    movel([0.093526, -1.335742, -2.600974, -0.775673, 1.570796, 1.664322],accel_mss,speed_ms,0,blend_radius_m)
    movel([0.093093, -1.336352, -2.600581, -0.775456, 1.570796, 1.663890],accel_mss,speed_ms,0,blend_radius_m)
    movel([0.092892, -1.336973, -2.600181, -0.775235, 1.570796, 1.663688],accel_mss,speed_ms,0,blend_radius_m)
    movel([0.091818, -1.346006, -2.594298, -0.772085, 1.570796, 1.662615],accel_mss,speed_ms,0,blend_radius_m)
    movel([0.090858, -1.354768, -2.588485, -0.769136, 1.570796, 1.661654],accel_mss,speed_ms,0,blend_radius_m)
    movel([0.090901, -1.355470, -2.588015, -0.768904, 1.570796, 1.661698],accel_mss,speed_ms,0,blend_radius_m)
    movel([0.091183, -1.356047, -2.587628, -0.768714, 1.570796, 1.661979],accel_mss,speed_ms,0,blend_radius_m)
    movel([0.091406, -1.356179, -2.587539, -0.768671, 1.570796, 1.662202],accel_mss,speed_ms,0,blend_radius_m)
    movel([0.091721, -1.356174, -2.587542, -0.768673, 1.570796, 1.662517],accel_mss,speed_ms,0,blend_radius_m)
    movel([0.094111, -1.355583, -2.587939, -0.768867, 1.570796, 1.664908],accel_mss,speed_ms,0,blend_radius_m)
    movel([0.104155, -1.352656, -2.589896, -0.769837, 1.570796, 1.674951],accel_mss,speed_ms,0,blend_radius_m)
    movel([0.116814, -1.348919, -2.592378, -0.771092, 1.570796, 1.687610],accel_mss,speed_ms,0,blend_radius_m)
    movel([0.119225, -1.332381, -2.603128, -0.776879, 1.570796, 1.690022],accel_mss,speed_ms,0,blend_radius_m)
    movel([0.119516, -1.329656, -2.604864, -0.777869, 1.570796, 1.690312],accel_mss,speed_ms,0,blend_radius_m)
    movel([0.119518, -1.328189, -2.605795, -0.778406, 1.570796, 1.690314],accel_mss,speed_ms,0,blend_radius_m)
    movel([0.119398, -1.327925, -2.605961, -0.778502, 1.570796, 1.690195],accel_mss,speed_ms,0,blend_radius_m)
    movel([0.119109, -1.327817, -2.606030, -0.778542, 1.570796, 1.689905],accel_mss,speed_ms,0,blend_radius_m)
    movel([0.118012, -1.327865, -2.606000, -0.778525, 1.570796, 1.688809],accel_mss,speed_ms,0,blend_radius_m)
    movel([0.116851, -1.328114, -2.605842, -0.778433, 1.570796, 1.687647],accel_mss,speed_ms,0,blend_radius_m)
    movel([0.116553, -1.328203, -2.605786, -0.778400, 1.570796, 1.687349],accel_mss,speed_ms,0,blend_radius_m)
    speed_ms = 0.005
    movel([0.116553, -1.319188, -2.601551, -0.791650, 1.570796, 1.687349],accel_mss,speed_ms,0,blend_radius_m)
    speed_ms = 0.040
    movel([0.074162, -1.348204, -2.582858, -0.781327, 1.570796, 1.644958],accel_mss,speed_ms,0,blend_radius_m)
    speed_ms = 0.005
    movel([0.074162, -1.357034, -2.586964, -0.768391, 1.570796, 1.644958],accel_mss,speed_ms,0,blend_radius_m)
    speed_ms = 0.035
    movel([0.079007, -1.355499, -2.587996, -0.768895, 1.570796, 1.649804],accel_mss,speed_ms,0,blend_radius_m)
    movel([0.085319, -1.353347, -2.589435, -0.769607, 1.570796, 1.656115],accel_mss,speed_ms,0,blend_radius_m)
    movel([0.085564, -1.353072, -2.589619, -0.769698, 1.570796, 1.656361],accel_mss,speed_ms,0,blend_radius_m)
    movel([0.085360, -1.352935, -2.589710, -0.769744, 1.570796, 1.656156],accel_mss,speed_ms,0,blend_radius_m)
    movel([0.082622, -1.353653, -2.589231, -0.769505, 1.570796, 1.653419],accel_mss,speed_ms,0,blend_radius_m)
    movel([0.074238, -1.356146, -2.587561, -0.768682, 1.570796, 1.645035],accel_mss,speed_ms,0,blend_radius_m)
    movel([0.069395, -1.357699, -2.586517, -0.768173, 1.570796, 1.640191],accel_mss,speed_ms,0,blend_radius_m)
    movel([0.063113, -1.359909, -2.585025, -0.767456, 1.570796, 1.633909],accel_mss,speed_ms,0,blend_radius_m)
    movel([0.062874, -1.360183, -2.584839, -0.767367, 1.570796, 1.633671],accel_mss,speed_ms,0,blend_radius_m)
    movel([0.063083, -1.360314, -2.584750, -0.767325, 1.570796, 1.633879],accel_mss,speed_ms,0,blend_radius_m)
    movel([0.065805, -1.359563, -2.585258, -0.767567, 1.570796, 1.636602],accel_mss,speed_ms,0,blend_radius_m)
    movel([0.074162, -1.357034, -2.586964, -0.768391, 1.570796, 1.644958],accel_mss,speed_ms,0,blend_radius_m)
    movel([0.076741, -1.356216, -2.587514, -0.768659, 1.570796, 1.647537],accel_mss,speed_ms,0,blend_radius_m)
    speed_ms = 0.005
    movel([0.076741, -1.347380, -2.583404, -0.781604, 1.570796, 1.647537],accel_mss,speed_ms,0,blend_radius_m)
    speed_ms = 0.040
    movel([0.074315, -1.346414, -2.584044, -0.781931, 1.570796, 1.645111],accel_mss,speed_ms,0,blend_radius_m)
    speed_ms = 0.005
    movel([0.074315, -1.355256, -2.588158, -0.768975, 1.570796, 1.645111],accel_mss,speed_ms,0,blend_radius_m)
    speed_ms = 0.035
    movel([0.065941, -1.357797, -2.586451, -0.768141, 1.570796, 1.636738],accel_mss,speed_ms,0,blend_radius_m)
    movel([0.063213, -1.358551, -2.585942, -0.767896, 1.570796, 1.634009],accel_mss,speed_ms,0,blend_radius_m)
    movel([0.063004, -1.358420, -2.586030, -0.767938, 1.570796, 1.633800],accel_mss,speed_ms,0,blend_radius_m)
    movel([0.063243, -1.358145, -2.586216, -0.768028, 1.570796, 1.634039],accel_mss,speed_ms,0,blend_radius_m)
    movel([0.069538, -1.355925, -2.587709, -0.768754, 1.570796, 1.640335],accel_mss,speed_ms,0,blend_radius_m)
    movel([0.074392, -1.354365, -2.588755, -0.769269, 1.570796, 1.645188],accel_mss,speed_ms,0,blend_radius_m)
    movel([0.082794, -1.351860, -2.590426, -0.770103, 1.570796, 1.653590],accel_mss,speed_ms,0,blend_radius_m)
    movel([0.085537, -1.351138, -2.590906, -0.770345, 1.570796, 1.656334],accel_mss,speed_ms,0,blend_radius_m)
    movel([0.085742, -1.351276, -2.590815, -0.770298, 1.570796, 1.656539],accel_mss,speed_ms,0,blend_radius_m)
    movel([0.085496, -1.351552, -2.590631, -0.770206, 1.570796, 1.656293],accel_mss,speed_ms,0,blend_radius_m)
    movel([0.079171, -1.353713, -2.589191, -0.769485, 1.570796, 1.649968],accel_mss,speed_ms,0,blend_radius_m)
    movel([0.074315, -1.355256, -2.588158, -0.768975, 1.570796, 1.645111],accel_mss,speed_ms,0,blend_radius_m)
    movel([0.071737, -1.356033, -2.587637, -0.768719, 1.570796, 1.642533],accel_mss,speed_ms,0,blend_radius_m)
    speed_ms = 0.005
    movel([0.071737, -1.347197, -2.583526, -0.781666, 1.570796, 1.642533],accel_mss,speed_ms,0,blend_radius_m)
    speed_ms = 0.040
    movel([0.074469, -1.344619, -2.585229, -0.782541, 1.570796, 1.645266],accel_mss,speed_ms,0,blend_radius_m)
    speed_ms = 0.005
    movel([0.074469, -1.353473, -2.589351, -0.769565, 1.570796, 1.645266],accel_mss,speed_ms,0,blend_radius_m)
    speed_ms = 0.035
    movel([0.067160, -1.355775, -2.587810, -0.768804, 1.570796, 1.637956],accel_mss,speed_ms,0,blend_radius_m)
    movel([0.064659, -1.356475, -2.587340, -0.768574, 1.570796, 1.635455],accel_mss,speed_ms,0,blend_radius_m)
    movel([0.063521, -1.356595, -2.587260, -0.768535, 1.570796, 1.634318],accel_mss,speed_ms,0,blend_radius_m)
    movel([0.063250, -1.356481, -2.587336, -0.768572, 1.570796, 1.634047],accel_mss,speed_ms,0,blend_radius_m)
    movel([0.063167, -1.356210, -2.587518, -0.768661, 1.570796, 1.633963],accel_mss,speed_ms,0,blend_radius_m)
    movel([0.063295, -1.355870, -2.587746, -0.768772, 1.570796, 1.634092],accel_mss,speed_ms,0,blend_radius_m)
    movel([0.063597, -1.355572, -2.587947, -0.768871, 1.570796, 1.634394],accel_mss,speed_ms,0,blend_radius_m)
    movel([0.064774, -1.354945, -2.588366, -0.769077, 1.570796, 1.635570],accel_mss,speed_ms,0,blend_radius_m)
    movel([0.067296, -1.354033, -2.588977, -0.769379, 1.570796, 1.638093],accel_mss,speed_ms,0,blend_radius_m)
    movel([0.074624, -1.351685, -2.590543, -0.770161, 1.570796, 1.645420],accel_mss,speed_ms,0,blend_radius_m)
    movel([0.081965, -1.349403, -2.592057, -0.770929, 1.570796, 1.652762],accel_mss,speed_ms,0,blend_radius_m)
    movel([0.084482, -1.348726, -2.592505, -0.771158, 1.570796, 1.655279],accel_mss,speed_ms,0,blend_radius_m)
    movel([0.085622, -1.348624, -2.592572, -0.771192, 1.570796, 1.656418],accel_mss,speed_ms,0,blend_radius_m)
    movel([0.085890, -1.348745, -2.592492, -0.771151, 1.570796, 1.656686],accel_mss,speed_ms,0,blend_radius_m)
    movel([0.085966, -1.349024, -2.592308, -0.771057, 1.570796, 1.656762],accel_mss,speed_ms,0,blend_radius_m)
    movel([0.085828, -1.349368, -2.592081, -0.770941, 1.570796, 1.656625],accel_mss,speed_ms,0,blend_radius_m)
    movel([0.085519, -1.349666, -2.591883, -0.770840, 1.570796, 1.656315],accel_mss,speed_ms,0,blend_radius_m)
    movel([0.084331, -1.350281, -2.591475, -0.770633, 1.570796, 1.655127],accel_mss,speed_ms,0,blend_radius_m)
    movel([0.081798, -1.351166, -2.590888, -0.770335, 1.570796, 1.652595],accel_mss,speed_ms,0,blend_radius_m)
    movel([0.074469, -1.353473, -2.589351, -0.769565, 1.570796, 1.645266],accel_mss,speed_ms,0,blend_radius_m)
    movel([0.071883, -1.354283, -2.588810, -0.769296, 1.570796, 1.642679],accel_mss,speed_ms,0,blend_radius_m)
    speed_ms = 0.005
    movel([0.071883, -1.345435, -2.584691, -0.782263, 1.570796, 1.642679],accel_mss,speed_ms,0,blend_radius_m)
    speed_ms = 0.040
    movel([0.075000, -1.341384, -2.587354, -0.783651, 1.570796, 1.645797],accel_mss,speed_ms,0,blend_radius_m)
    speed_ms = 0.005
    movel([0.075000, -1.350258, -2.591490, -0.770640, 1.570796, 1.645797],accel_mss,speed_ms,0,blend_radius_m)
    speed_ms = 0.035
    movel([0.062813, -1.354160, -2.588892, -0.769337, 1.570796, 1.633609],accel_mss,speed_ms,0,blend_radius_m)
    movel([0.063322, -1.347243, -2.593484, -0.771662, 1.570796, 1.634118],accel_mss,speed_ms,0,blend_radius_m)
    movel([0.063839, -1.340253, -2.598058, -0.774078, 1.570796, 1.634635],accel_mss,speed_ms,0,blend_radius_m)
    movel([0.076231, -1.336205, -2.600676, -0.775508, 1.570796, 1.647027],accel_mss,speed_ms,0,blend_radius_m)
    movel([0.088671, -1.332244, -2.603216, -0.776929, 1.570796, 1.659467],accel_mss,speed_ms,0,blend_radius_m)
    movel([0.087946, -1.339382, -2.598623, -0.774384, 1.570796, 1.658742],accel_mss,speed_ms,0,blend_radius_m)
    movel([0.087233, -1.346443, -2.594011, -0.771935, 1.570796, 1.658029],accel_mss,speed_ms,0,blend_radius_m)
    movel([0.075000, -1.350258, -2.591490, -0.770640, 1.570796, 1.645797],accel_mss,speed_ms,0,blend_radius_m)
    movel([0.072403, -1.351082, -2.590944, -0.770364, 1.570796, 1.643200],accel_mss,speed_ms,0,blend_radius_m)
    speed_ms = 0.005
    movel([0.072403, -1.342212, -2.586811, -0.783366, 1.570796, 1.643200],accel_mss,speed_ms,0,blend_radius_m)
    speed_ms = 0.040
    movel([0.069921, -1.327417, -2.596364, -0.788608, 1.570796, 1.640717],accel_mss,speed_ms,0,blend_radius_m)
    speed_ms = 0.005
    movel([0.069921, -1.336381, -2.600563, -0.775446, 1.570796, 1.640717],accel_mss,speed_ms,0,blend_radius_m)
    speed_ms = 0.035
    movel([0.075354, -1.334483, -2.601783, -0.776123, 1.570796, 1.646150],accel_mss,speed_ms,0,blend_radius_m)
    movel([0.076046, -1.328181, -2.605800, -0.778409, 1.570796, 1.646843],accel_mss,speed_ms,0,blend_radius_m)
    movel([0.076292, -1.325734, -2.607345, -0.779310, 1.570796, 1.647089],accel_mss,speed_ms,0,blend_radius_m)
    movel([0.076527, -1.321857, -2.609777, -0.780755, 1.570796, 1.647323],accel_mss,speed_ms,0,blend_radius_m)
    movel([0.076407, -1.321615, -2.609928, -0.780846, 1.570796, 1.647203],accel_mss,speed_ms,0,blend_radius_m)
    movel([0.076099, -1.321589, -2.609944, -0.780856, 1.570796, 1.646895],accel_mss,speed_ms,0,blend_radius_m)
    movel([0.074610, -1.321987, -2.609696, -0.780707, 1.570796, 1.645406],accel_mss,speed_ms,0,blend_radius_m)
    movel([0.070780, -1.323169, -2.608956, -0.780264, 1.570796, 1.641576],accel_mss,speed_ms,0,blend_radius_m)
    movel([0.065505, -1.324941, -2.607844, -0.779604, 1.570796, 1.636301],accel_mss,speed_ms,0,blend_radius_m)
    movel([0.064998, -1.331651, -2.603594, -0.777144, 1.570796, 1.635794],accel_mss,speed_ms,0,blend_radius_m)
    movel([0.064499, -1.338294, -2.599328, -0.774768, 1.570796, 1.635295],accel_mss,speed_ms,0,blend_radius_m)
    movel([0.069921, -1.336381, -2.600563, -0.775446, 1.570796, 1.640717],accel_mss,speed_ms,0,blend_radius_m)
    movel([0.072570, -1.335452, -2.601160, -0.775777, 1.570796, 1.643366],accel_mss,speed_ms,0,blend_radius_m)
    speed_ms = 0.005
    movel([0.072570, -1.326483, -2.596958, -0.788949, 1.570796, 1.643366],accel_mss,speed_ms,0,blend_radius_m)
    speed_ms = 0.040
    movel([0.082365, -1.323365, -2.598930, -0.790095, 1.570796, 1.653161],accel_mss,speed_ms,0,blend_radius_m)
    speed_ms = 0.005
    movel([0.082365, -1.332354, -2.603146, -0.776889, 1.570796, 1.653161],accel_mss,speed_ms,0,blend_radius_m)
    speed_ms = 0.035
    movel([0.087793, -1.330758, -2.604164, -0.777468, 1.570796, 1.658590],accel_mss,speed_ms,0,blend_radius_m)
    movel([0.088479, -1.323981, -2.608447, -0.779961, 1.570796, 1.659275],accel_mss,speed_ms,0,blend_radius_m)
    movel([0.089175, -1.317133, -2.612713, -0.782543, 1.570796, 1.659971],accel_mss,speed_ms,0,blend_radius_m)
    movel([0.083497, -1.318972, -2.611573, -0.781844, 1.570796, 1.654293],accel_mss,speed_ms,0,blend_radius_m)
    movel([0.077826, -1.320830, -2.610417, -0.781141, 1.570796, 1.648622],accel_mss,speed_ms,0,blend_radius_m)
    movel([0.077382, -1.327431, -2.606274, -0.778684, 1.570796, 1.648179],accel_mss,speed_ms,0,blend_radius_m)
    movel([0.076943, -1.333968, -2.602113, -0.776308, 1.570796, 1.647739],accel_mss,speed_ms,0,blend_radius_m)
    movel([0.082365, -1.332354, -2.603146, -0.776889, 1.570796, 1.653161],accel_mss,speed_ms,0,blend_radius_m)
    movel([0.085012, -1.331573, -2.603644, -0.777172, 1.570796, 1.655808],accel_mss,speed_ms,0,blend_radius_m)
    speed_ms = 0.005
    movel([0.085012, -1.322579, -2.599424, -0.790385, 1.570796, 1.655808],accel_mss,speed_ms,0,blend_radius_m)
    speed_ms = 0.040
    movel([0.113728, -1.302056, -2.612063, -0.798270, 1.570796, 1.684524],accel_mss,speed_ms,0,blend_radius_m)
    speed_ms = 0.005
    movel([0.113728, -1.311174, -2.616374, -0.784841, 1.570796, 1.684524],accel_mss,speed_ms,0,blend_radius_m)
    speed_ms = 0.035
    movel([0.134816, -1.304786, -2.620247, -0.787356, 1.570796, 1.705613],accel_mss,speed_ms,0,blend_radius_m)
    movel([0.138512, -1.281408, -2.633973, -0.797009, 1.570796, 1.709308],accel_mss,speed_ms,0,blend_radius_m)
    movel([0.142413, -1.257135, -2.647496, -0.807758, 1.570796, 1.713209],accel_mss,speed_ms,0,blend_radius_m)
    movel([0.120006, -1.264267, -2.643598, -0.804524, 1.570796, 1.690802],accel_mss,speed_ms,0,blend_radius_m)
    movel([0.097729, -1.271692, -2.639473, -0.801224, 1.570796, 1.668525],accel_mss,speed_ms,0,blend_radius_m)
    movel([0.095175, -1.295169, -2.625978, -0.791242, 1.570796, 1.665971],accel_mss,speed_ms,0,blend_radius_m)
    movel([0.092754, -1.317830, -2.612282, -0.782278, 1.570796, 1.663550],accel_mss,speed_ms,0,blend_radius_m)
    movel([0.113728, -1.311174, -2.616374, -0.784841, 1.570796, 1.684524],accel_mss,speed_ms,0,blend_radius_m)
    movel([0.116442, -1.310336, -2.616885, -0.785168, 1.570796, 1.687239],accel_mss,speed_ms,0,blend_radius_m)
    speed_ms = 0.005
    movel([0.116442, -1.301214, -2.612570, -0.798605, 1.570796, 1.687239],accel_mss,speed_ms,0,blend_radius_m)
    speed_ms = 0.040
    movel([0.120277, -1.252809, -2.640206, -0.819374, 1.570796, 1.691073],accel_mss,speed_ms,0,blend_radius_m)
    speed_ms = 0.005
    movel([0.120277, -1.262191, -2.644739, -0.805459, 1.570796, 1.691073],accel_mss,speed_ms,0,blend_radius_m)
    speed_ms = 0.035
    movel([0.129753, -1.259094, -2.646431, -0.806863, 1.570796, 1.700549],accel_mss,speed_ms,0,blend_radius_m)
    movel([0.141933, -1.255007, -2.648648, -0.808735, 1.570796, 1.712729],accel_mss,speed_ms,0,blend_radius_m)
    movel([0.142238, -1.254672, -2.648828, -0.808889, 1.570796, 1.713034],accel_mss,speed_ms,0,blend_radius_m)
    movel([0.142012, -1.254503, -2.648919, -0.808967, 1.570796, 1.712808],accel_mss,speed_ms,0,blend_radius_m)
    movel([0.136669, -1.256047, -2.648086, -0.808257, 1.570796, 1.707466],accel_mss,speed_ms,0,blend_radius_m)
    movel([0.120416, -1.261150, -2.645309, -0.805930, 1.570796, 1.691212],accel_mss,speed_ms,0,blend_radius_m)
    movel([0.110953, -1.264308, -2.643575, -0.804506, 1.570796, 1.681749],accel_mss,speed_ms,0,blend_radius_m)
    movel([0.098869, -1.268617, -2.641190, -0.802582, 1.570796, 1.669665],accel_mss,speed_ms,0,blend_radius_m)
    movel([0.098580, -1.268949, -2.641005, -0.802435, 1.570796, 1.669376],accel_mss,speed_ms,0,blend_radius_m)
    movel([0.098815, -1.269102, -2.640919, -0.802367, 1.570796, 1.669612],accel_mss,speed_ms,0,blend_radius_m)
    movel([0.104107, -1.267439, -2.641844, -0.803106, 1.570796, 1.674903],accel_mss,speed_ms,0,blend_radius_m)
    movel([0.120277, -1.262191, -2.644739, -0.805459, 1.570796, 1.691073],accel_mss,speed_ms,0,blend_radius_m)
    movel([0.123150, -1.261245, -2.645257, -0.805887, 1.570796, 1.693947],accel_mss,speed_ms,0,blend_radius_m)
    speed_ms = 0.005
    movel([0.123150, -1.251858, -2.640720, -0.819811, 1.570796, 1.693947],accel_mss,speed_ms,0,blend_radius_m)
    speed_ms = 0.040
    movel([0.120555, -1.250715, -2.641337, -0.820337, 1.570796, 1.691351],accel_mss,speed_ms,0,blend_radius_m)
    speed_ms = 0.005
    movel([0.120555, -1.260107, -2.645879, -0.806403, 1.570796, 1.691351],accel_mss,speed_ms,0,blend_radius_m)
    speed_ms = 0.035
    movel([0.142487, -1.253079, -2.649686, -0.809624, 1.570796, 1.713283],accel_mss,speed_ms,0,blend_radius_m)
    movel([0.142694, -1.251749, -2.650399, -0.810241, 1.570796, 1.713491],accel_mss,speed_ms,0,blend_radius_m)
    movel([0.142903, -1.250416, -2.651113, -0.810861, 1.570796, 1.713699],accel_mss,speed_ms,0,blend_radius_m)
    movel([0.120905, -1.257492, -2.647302, -0.807594, 1.570796, 1.691701],accel_mss,speed_ms,0,blend_radius_m)
    movel([0.099033, -1.264850, -2.643276, -0.804263, 1.570796, 1.669830],accel_mss,speed_ms,0,blend_radius_m)
    movel([0.098891, -1.266134, -2.642567, -0.803688, 1.570796, 1.669687],accel_mss,speed_ms,0,blend_radius_m)
    movel([0.098749, -1.267415, -2.641857, -0.803117, 1.570796, 1.669546],accel_mss,speed_ms,0,blend_radius_m)
    movel([0.120555, -1.260107, -2.645879, -0.806403, 1.570796, 1.691351],accel_mss,speed_ms,0,blend_radius_m)
    movel([0.123434, -1.259166, -2.646392, -0.806831, 1.570796, 1.694230],accel_mss,speed_ms,0,blend_radius_m)
    speed_ms = 0.005
    movel([0.123434, -1.249769, -2.641846, -0.820774, 1.570796, 1.694230],accel_mss,speed_ms,0,blend_radius_m)
    speed_ms = 0.040
    movel([0.121045, -1.247034, -2.643312, -0.822044, 1.570796, 1.691842],accel_mss,speed_ms,0,blend_radius_m)
    speed_ms = 0.005
    movel([0.121045, -1.256443, -2.647871, -0.808075, 1.570796, 1.691842],accel_mss,speed_ms,0,blend_radius_m)
    speed_ms = 0.035
    movel([0.135426, -1.251755, -2.650396, -0.810238, 1.570796, 1.706223],accel_mss,speed_ms,0,blend_radius_m)
    movel([0.140187, -1.250123, -2.651269, -0.810997, 1.570796, 1.710984],accel_mss,speed_ms,0,blend_radius_m)
    movel([0.142550, -1.249119, -2.651804, -0.811466, 1.570796, 1.713347],accel_mss,speed_ms,0,blend_radius_m)
    movel([0.143005, -1.248755, -2.651998, -0.811636, 1.570796, 1.713802],accel_mss,speed_ms,0,blend_radius_m)
    movel([0.143238, -1.248277, -2.652252, -0.811860, 1.570796, 1.714034],accel_mss,speed_ms,0,blend_radius_m)
    movel([0.143139, -1.247903, -2.652451, -0.812035, 1.570796, 1.713935],accel_mss,speed_ms,0,blend_radius_m)
    movel([0.142756, -1.247802, -2.652504, -0.812082, 1.570796, 1.713552],accel_mss,speed_ms,0,blend_radius_m)
    movel([0.140472, -1.248269, -2.652257, -0.811864, 1.570796, 1.711269],accel_mss,speed_ms,0,blend_radius_m)
    movel([0.135738, -1.249663, -2.651514, -0.811212, 1.570796, 1.706534],accel_mss,speed_ms,0,blend_radius_m)
    movel([0.121327, -1.254340, -2.649007, -0.809042, 1.570796, 1.692123],accel_mss,speed_ms,0,blend_radius_m)
    movel([0.106966, -1.259175, -2.646388, -0.806827, 1.570796, 1.677763],accel_mss,speed_ms,0,blend_radius_m)
    movel([0.102241, -1.260904, -2.645444, -0.806041, 1.570796, 1.673038],accel_mss,speed_ms,0,blend_radius_m)
    movel([0.099911, -1.261956, -2.644868, -0.805565, 1.570796, 1.670707],accel_mss,speed_ms,0,blend_radius_m)
    movel([0.099472, -1.262324, -2.644666, -0.805399, 1.570796, 1.670268],accel_mss,speed_ms,0,blend_radius_m)
    movel([0.099262, -1.262791, -2.644410, -0.805189, 1.570796, 1.670058],accel_mss,speed_ms,0,blend_radius_m)
    movel([0.099380, -1.263144, -2.644216, -0.805029, 1.570796, 1.670177],accel_mss,speed_ms,0,blend_radius_m)
    movel([0.099769, -1.263226, -2.644171, -0.804992, 1.570796, 1.670566],accel_mss,speed_ms,0,blend_radius_m)
    movel([0.102037, -1.262698, -2.644461, -0.805230, 1.570796, 1.672833],accel_mss,speed_ms,0,blend_radius_m)
    movel([0.106723, -1.261215, -2.645273, -0.805900, 1.570796, 1.677520],accel_mss,speed_ms,0,blend_radius_m)
    movel([0.121045, -1.256443, -2.647871, -0.808075, 1.570796, 1.691842],accel_mss,speed_ms,0,blend_radius_m)
    movel([0.123937, -1.255490, -2.648386, -0.808512, 1.570796, 1.694733],accel_mss,speed_ms,0,blend_radius_m)
    speed_ms = 0.005
    movel([0.123937, -1.246076, -2.643823, -0.822490, 1.570796, 1.694733],accel_mss,speed_ms,0,blend_radius_m)
    speed_ms = 0.040
    movel([0.121469, -1.243862, -2.645001, -0.823527, 1.570796, 1.692265],accel_mss,speed_ms,0,blend_radius_m)
    speed_ms = 0.005
    movel([0.121469, -1.253286, -2.649574, -0.809529, 1.570796, 1.692265],accel_mss,speed_ms,0,blend_radius_m)
    speed_ms = 0.035
    movel([0.105133, -1.258657, -2.646669, -0.807062, 1.570796, 1.675929],accel_mss,speed_ms,0,blend_radius_m)
    movel([0.099787, -1.260361, -2.645740, -0.806287, 1.570796, 1.670583],accel_mss,speed_ms,0,blend_radius_m)
    movel([0.099549, -1.260207, -2.645825, -0.806357, 1.570796, 1.670346],accel_mss,speed_ms,0,blend_radius_m)
    movel([0.099842, -1.259869, -2.646009, -0.806511, 1.570796, 1.670638],accel_mss,speed_ms,0,blend_radius_m)
    movel([0.112050, -1.255462, -2.648402, -0.808526, 1.570796, 1.682846],accel_mss,speed_ms,0,blend_radius_m)
    movel([0.121610, -1.252230, -2.650141, -0.810018, 1.570796, 1.692407],accel_mss,speed_ms,0,blend_radius_m)
    movel([0.138032, -1.247004, -2.652928, -0.812457, 1.570796, 1.708829],accel_mss,speed_ms,0,blend_radius_m)
    movel([0.143430, -1.245422, -2.653765, -0.813202, 1.570796, 1.714226],accel_mss,speed_ms,0,blend_radius_m)
    movel([0.143659, -1.245593, -2.653675, -0.813121, 1.570796, 1.714455],accel_mss,speed_ms,0,blend_radius_m)
    movel([0.143350, -1.245933, -2.653495, -0.812961, 1.570796, 1.714146],accel_mss,speed_ms,0,blend_radius_m)
    movel([0.131042, -1.250116, -2.651272, -0.811000, 1.570796, 1.701839],accel_mss,speed_ms,0,blend_radius_m)
    movel([0.121469, -1.253286, -2.649574, -0.809529, 1.570796, 1.692265],accel_mss,speed_ms,0,blend_radius_m)
    movel([0.118572, -1.254225, -2.649069, -0.809095, 1.570796, 1.689369],accel_mss,speed_ms,0,blend_radius_m)
    speed_ms = 0.005
    movel([0.118572, -1.244805, -2.644500, -0.823084, 1.570796, 1.689369],accel_mss,speed_ms,0,blend_radius_m)
    speed_ms = 0.040
    movel([0.121895, -1.240674, -2.646686, -0.825029, 1.570796, 1.692691],accel_mss,speed_ms,0,blend_radius_m)
    speed_ms = 0.005
    movel([0.121895, -1.250113, -2.651274, -0.811002, 1.570796, 1.692691],accel_mss,speed_ms,0,blend_radius_m)
    speed_ms = 0.035
    movel([0.099260, -1.257814, -2.647128, -0.807447, 1.570796, 1.670056],accel_mss,speed_ms,0,blend_radius_m)
    movel([0.101199, -1.240438, -2.656383, -0.815568, 1.570796, 1.671995],accel_mss,speed_ms,0,blend_radius_m)
    movel([0.103217, -1.222583, -2.665523, -0.824283, 1.570796, 1.674013],accel_mss,speed_ms,0,blend_radius_m)
    movel([0.126797, -1.214135, -2.669720, -0.828534, 1.570796, 1.697593],accel_mss,speed_ms,0,blend_radius_m)
    movel([0.150532, -1.206002, -2.673684, -0.832703, 1.570796, 1.721329],accel_mss,speed_ms,0,blend_radius_m)
    movel([0.147540, -1.224622, -2.664498, -0.823269, 1.570796, 1.718336],accel_mss,speed_ms,0,blend_radius_m)
    movel([0.144667, -1.242712, -2.655192, -0.814485, 1.570796, 1.715464],accel_mss,speed_ms,0,blend_radius_m)
    movel([0.121895, -1.250113, -2.651274, -0.811002, 1.570796, 1.692691],accel_mss,speed_ms,0,blend_radius_m)
    movel([0.118985, -1.251084, -2.650755, -0.810550, 1.570796, 1.689781],accel_mss,speed_ms,0,blend_radius_m)
    speed_ms = 0.005
    movel([0.118985, -1.241650, -2.646172, -0.824568, 1.570796, 1.689781],accel_mss,speed_ms,0,blend_radius_m)
    speed_ms = 0.040
    movel([0.126726, -1.202963, -2.665736, -0.843690, 1.570796, 1.697522],accel_mss,speed_ms,0,blend_radius_m)
    speed_ms = 0.005
    movel([0.126726, -1.212558, -2.670494, -0.829337, 1.570796, 1.697522],accel_mss,speed_ms,0,blend_radius_m)
    speed_ms = 0.035
    movel([0.149588, -1.204692, -2.674316, -0.833381, 1.570796, 1.720384],accel_mss,speed_ms,0,blend_radius_m)
    movel([0.151219, -1.194576, -2.679130, -0.838683, 1.570796, 1.722015],accel_mss,speed_ms,0,blend_radius_m)
    movel([0.152886, -1.184296, -2.683908, -0.844185, 1.570796, 1.723683],accel_mss,speed_ms,0,blend_radius_m)
    movel([0.129497, -1.192581, -2.680066, -0.839742, 1.570796, 1.700293],accel_mss,speed_ms,0,blend_radius_m)
    movel([0.106263, -1.201163, -2.676008, -0.835218, 1.570796, 1.677059],accel_mss,speed_ms,0,blend_radius_m)
    movel([0.105123, -1.211012, -2.671251, -0.830126, 1.570796, 1.675919],accel_mss,speed_ms,0,blend_radius_m)
    movel([0.104008, -1.220714, -2.666458, -0.825217, 1.570796, 1.674804],accel_mss,speed_ms,0,blend_radius_m)
    movel([0.126726, -1.212558, -2.670494, -0.829337, 1.570796, 1.697522],accel_mss,speed_ms,0,blend_radius_m)
    movel([0.129766, -1.211492, -2.671016, -0.829881, 1.570796, 1.700562],accel_mss,speed_ms,0,blend_radius_m)
    speed_ms = 0.005
    movel([0.129766, -1.201893, -2.666253, -0.844243, 1.570796, 1.700562],accel_mss,speed_ms,0,blend_radius_m)
    speed_ms = 0.040
    movel([0.178723, -1.185527, -2.674008, -0.852854, 1.570796, 1.749519],accel_mss,speed_ms,0,blend_radius_m)
    speed_ms = 0.005
    movel([0.178723, -1.195182, -2.678844, -0.838362, 1.570796, 1.749519],accel_mss,speed_ms,0,blend_radius_m)
    speed_ms = 0.035
    movel([0.201836, -1.188058, -2.682172, -0.842158, 1.570796, 1.772633],accel_mss,speed_ms,0,blend_radius_m)
    movel([0.204073, -1.177494, -2.687007, -0.847888, 1.570796, 1.774869],accel_mss,speed_ms,0,blend_radius_m)
    movel([0.206362, -1.166750, -2.691803, -0.853836, 1.570796, 1.777158],accel_mss,speed_ms,0,blend_radius_m)
    movel([0.182702, -1.174269, -2.688459, -0.849661, 1.570796, 1.753498],accel_mss,speed_ms,0,blend_radius_m)
    movel([0.159147, -1.182140, -2.684895, -0.845354, 1.570796, 1.729943],accel_mss,speed_ms,0,blend_radius_m)
    movel([0.157407, -1.192476, -2.680115, -0.839798, 1.570796, 1.728204],accel_mss,speed_ms,0,blend_radius_m)
    movel([0.155706, -1.202647, -2.675298, -0.834444, 1.570796, 1.726503],accel_mss,speed_ms,0,blend_radius_m)
    movel([0.178723, -1.195182, -2.678844, -0.838362, 1.570796, 1.749519],accel_mss,speed_ms,0,blend_radius_m)
    movel([0.181799, -1.194212, -2.679301, -0.838876, 1.570796, 1.752596],accel_mss,speed_ms,0,blend_radius_m)
    speed_ms = 0.005
    movel([0.181799, -1.184554, -2.674459, -0.853375, 1.570796, 1.752596],accel_mss,speed_ms,0,blend_radius_m)
    speed_ms = 0.040
    movel([0.170964, -1.224975, -2.654814, -0.832601, 1.570796, 1.741760],accel_mss,speed_ms,0,blend_radius_m)
    speed_ms = 0.005
    movel([0.170964, -1.234483, -2.659472, -0.818433, 1.570796, 1.741760],accel_mss,speed_ms,0,blend_radius_m)
    speed_ms = 0.035
    movel([0.193490, -1.228067, -2.662755, -0.821567, 1.570796, 1.764287],accel_mss,speed_ms,0,blend_radius_m)
    movel([0.197334, -1.209522, -2.671977, -0.830889, 1.570796, 1.768131],accel_mss,speed_ms,0,blend_radius_m)
    movel([0.199301, -1.199962, -2.676581, -0.835846, 1.570796, 1.770097],accel_mss,speed_ms,0,blend_radius_m)
    movel([0.200933, -1.190783, -2.680906, -0.840700, 1.570796, 1.771729],accel_mss,speed_ms,0,blend_radius_m)
    movel([0.200878, -1.190484, -2.681045, -0.840860, 1.570796, 1.771674],accel_mss,speed_ms,0,blend_radius_m)
    movel([0.200628, -1.190354, -2.681106, -0.840929, 1.570796, 1.771424],accel_mss,speed_ms,0,blend_radius_m)
    movel([0.200026, -1.190429, -2.681071, -0.840889, 1.570796, 1.770823],accel_mss,speed_ms,0,blend_radius_m)
    movel([0.177133, -1.197469, -2.677764, -0.837155, 1.570796, 1.747930],accel_mss,speed_ms,0,blend_radius_m)
    movel([0.154454, -1.204965, -2.674184, -0.833239, 1.570796, 1.725251],accel_mss,speed_ms,0,blend_radius_m)
    movel([0.151426, -1.223361, -2.665132, -0.823896, 1.570796, 1.722223],accel_mss,speed_ms,0,blend_radius_m)
    movel([0.148519, -1.241238, -2.655965, -0.815186, 1.570796, 1.719315],accel_mss,speed_ms,0,blend_radius_m)
    movel([0.170964, -1.234483, -2.659472, -0.818433, 1.570796, 1.741760],accel_mss,speed_ms,0,blend_radius_m)
    movel([0.173904, -1.233625, -2.659914, -0.818850, 1.570796, 1.744701],accel_mss,speed_ms,0,blend_radius_m)
    speed_ms = 0.005
    movel([0.173904, -1.224113, -2.655251, -0.833024, 1.570796, 1.744701],accel_mss,speed_ms,0,blend_radius_m)
    speed_ms = 0.040
    movel([0.170186, -1.228469, -2.653029, -0.830891, 1.570796, 1.740982],accel_mss,speed_ms,0,blend_radius_m)
    speed_ms = 0.005
    movel([0.170186, -1.237962, -2.657672, -0.816754, 1.570796, 1.740982],accel_mss,speed_ms,0,blend_radius_m)
    speed_ms = 0.035
    movel([0.182708, -1.234267, -2.659584, -0.818538, 1.570796, 1.753504],accel_mss,speed_ms,0,blend_radius_m)
    movel([0.188419, -1.232517, -2.660483, -0.819389, 1.570796, 1.759215],accel_mss,speed_ms,0,blend_radius_m)
    movel([0.191800, -1.231374, -2.661069, -0.819946, 1.570796, 1.762597],accel_mss,speed_ms,0,blend_radius_m)
    movel([0.192177, -1.231118, -2.661200, -0.820071, 1.570796, 1.762974],accel_mss,speed_ms,0,blend_radius_m)
    movel([0.192385, -1.230741, -2.661393, -0.820255, 1.570796, 1.763181],accel_mss,speed_ms,0,blend_radius_m)
    movel([0.192316, -1.230442, -2.661546, -0.820402, 1.570796, 1.763112],accel_mss,speed_ms,0,blend_radius_m)
    movel([0.192004, -1.230380, -2.661577, -0.820432, 1.570796, 1.762800],accel_mss,speed_ms,0,blend_radius_m)
    movel([0.188697, -1.231135, -2.661191, -0.820063, 1.570796, 1.759494],accel_mss,speed_ms,0,blend_radius_m)
    movel([0.183024, -1.232652, -2.660414, -0.819323, 1.570796, 1.753821],accel_mss,speed_ms,0,blend_radius_m)
    movel([0.170489, -1.236313, -2.658527, -0.817549, 1.570796, 1.741285],accel_mss,speed_ms,0,blend_radius_m)
    movel([0.157971, -1.240126, -2.656546, -0.815717, 1.570796, 1.728768],accel_mss,speed_ms,0,blend_radius_m)
    movel([0.152285, -1.241994, -2.655569, -0.814826, 1.570796, 1.723081],accel_mss,speed_ms,0,blend_radius_m)
    movel([0.148931, -1.243221, -2.654925, -0.814243, 1.570796, 1.719727],accel_mss,speed_ms,0,blend_radius_m)
    movel([0.148564, -1.243482, -2.654787, -0.814119, 1.570796, 1.719360],accel_mss,speed_ms,0,blend_radius_m)
    movel([0.148374, -1.243852, -2.654593, -0.813944, 1.570796, 1.719170],accel_mss,speed_ms,0,blend_radius_m)
    movel([0.148458, -1.244136, -2.654443, -0.813810, 1.570796, 1.719254],accel_mss,speed_ms,0,blend_radius_m)
    movel([0.148775, -1.244183, -2.654419, -0.813787, 1.570796, 1.719571],accel_mss,speed_ms,0,blend_radius_m)
    movel([0.152063, -1.243338, -2.654863, -0.814188, 1.570796, 1.722859],accel_mss,speed_ms,0,blend_radius_m)
    movel([0.157700, -1.241710, -2.655718, -0.814961, 1.570796, 1.728496],accel_mss,speed_ms,0,blend_radius_m)
    movel([0.170186, -1.237962, -2.657672, -0.816754, 1.570796, 1.740982],accel_mss,speed_ms,0,blend_radius_m)
    movel([0.173119, -1.237087, -2.658127, -0.817175, 1.570796, 1.743916],accel_mss,speed_ms,0,blend_radius_m)
    speed_ms = 0.005
    movel([0.173119, -1.227590, -2.653480, -0.831320, 1.570796, 1.743916],accel_mss,speed_ms,0,blend_radius_m)
    speed_ms = 0.040
    movel([0.169583, -1.231768, -2.651332, -0.829289, 1.570796, 1.740380],accel_mss,speed_ms,0,blend_radius_m)
    speed_ms = 0.005
    movel([0.169583, -1.241248, -2.655960, -0.815182, 1.570796, 1.740380],accel_mss,speed_ms,0,blend_radius_m)
    speed_ms = 0.035
    movel([0.155296, -1.245534, -2.653706, -0.813149, 1.570796, 1.726092],accel_mss,speed_ms,0,blend_radius_m)
    movel([0.150619, -1.246856, -2.653006, -0.812527, 1.570796, 1.721416],accel_mss,speed_ms,0,blend_radius_m)
    movel([0.148370, -1.247296, -2.652773, -0.812320, 1.570796, 1.719166],accel_mss,speed_ms,0,blend_radius_m)
    movel([0.147989, -1.247190, -2.652829, -0.812370, 1.570796, 1.718786],accel_mss,speed_ms,0,blend_radius_m)
    movel([0.147895, -1.246816, -2.653027, -0.812545, 1.570796, 1.718691],accel_mss,speed_ms,0,blend_radius_m)
    movel([0.148126, -1.246341, -2.653279, -0.812769, 1.570796, 1.718923],accel_mss,speed_ms,0,blend_radius_m)
    movel([0.148584, -1.245973, -2.653474, -0.812942, 1.570796, 1.719381],accel_mss,speed_ms,0,blend_radius_m)
    movel([0.150927, -1.244986, -2.653995, -0.813408, 1.570796, 1.721723],accel_mss,speed_ms,0,blend_radius_m)
    movel([0.155655, -1.243408, -2.654827, -0.814155, 1.570796, 1.726451],accel_mss,speed_ms,0,blend_radius_m)
    movel([0.169984, -1.239059, -2.657102, -0.816228, 1.570796, 1.740781],accel_mss,speed_ms,0,blend_radius_m)
    movel([0.184343, -1.234884, -2.659266, -0.818239, 1.570796, 1.755139],accel_mss,speed_ms,0,blend_radius_m)
    movel([0.189052, -1.233661, -2.659896, -0.818832, 1.570796, 1.759849],accel_mss,speed_ms,0,blend_radius_m)
    movel([0.191309, -1.233288, -2.660087, -0.819013, 1.570796, 1.762105],accel_mss,speed_ms,0,blend_radius_m)
    movel([0.191682, -1.233414, -2.660023, -0.818952, 1.570796, 1.762478],accel_mss,speed_ms,0,blend_radius_m)
    movel([0.191756, -1.233807, -2.659820, -0.818761, 1.570796, 1.762552],accel_mss,speed_ms,0,blend_radius_m)
    movel([0.191502, -1.234293, -2.659571, -0.818526, 1.570796, 1.762298],accel_mss,speed_ms,0,blend_radius_m)
    movel([0.191030, -1.234656, -2.659383, -0.818350, 1.570796, 1.761826],accel_mss,speed_ms,0,blend_radius_m)
    movel([0.188663, -1.235587, -2.658903, -0.817899, 1.570796, 1.759460],accel_mss,speed_ms,0,blend_radius_m)
    movel([0.183914, -1.237057, -2.658142, -0.817190, 1.570796, 1.754710],accel_mss,speed_ms,0,blend_radius_m)
    movel([0.169583, -1.241248, -2.655960, -0.815182, 1.570796, 1.740380],accel_mss,speed_ms,0,blend_radius_m)
    movel([0.166664, -1.242113, -2.655507, -0.814770, 1.570796, 1.737460],accel_mss,speed_ms,0,blend_radius_m)
    speed_ms = 0.005
    movel([0.166664, -1.232637, -2.650882, -0.828869, 1.570796, 1.737460],accel_mss,speed_ms,0,blend_radius_m)
    speed_ms = 0.040
    movel([0.168985, -1.235051, -2.649630, -0.827708, 1.570796, 1.739782],accel_mss,speed_ms,0,blend_radius_m)
    speed_ms = 0.005
    movel([0.168985, -1.244516, -2.654243, -0.813630, 1.570796, 1.739782],accel_mss,speed_ms,0,blend_radius_m)
    speed_ms = 0.035
    movel([0.183262, -1.240361, -2.656423, -0.815605, 1.570796, 1.754059],accel_mss,speed_ms,0,blend_radius_m)
    movel([0.187994, -1.238903, -2.657183, -0.816303, 1.570796, 1.758791],accel_mss,speed_ms,0,blend_radius_m)
    movel([0.190352, -1.237979, -2.657664, -0.816746, 1.570796, 1.761148],accel_mss,speed_ms,0,blend_radius_m)
    movel([0.190822, -1.237618, -2.657851, -0.816920, 1.570796, 1.761618],accel_mss,speed_ms,0,blend_radius_m)
    movel([0.191075, -1.237136, -2.658101, -0.817152, 1.570796, 1.761871],accel_mss,speed_ms,0,blend_radius_m)
    movel([0.191001, -1.236744, -2.658304, -0.817341, 1.570796, 1.761797],accel_mss,speed_ms,0,blend_radius_m)
    movel([0.190629, -1.236619, -2.658369, -0.817401, 1.570796, 1.761425],accel_mss,speed_ms,0,blend_radius_m)
    movel([0.188381, -1.236987, -2.658178, -0.817223, 1.570796, 1.759177],accel_mss,speed_ms,0,blend_radius_m)
    movel([0.183688, -1.238199, -2.657549, -0.816640, 1.570796, 1.754485],accel_mss,speed_ms,0,blend_radius_m)
    movel([0.169384, -1.242339, -2.655388, -0.814662, 1.570796, 1.740180],accel_mss,speed_ms,0,blend_radius_m)
    movel([0.155107, -1.246650, -2.653115, -0.812623, 1.570796, 1.725903],accel_mss,speed_ms,0,blend_radius_m)
    movel([0.150396, -1.248216, -2.652285, -0.811889, 1.570796, 1.721192],accel_mss,speed_ms,0,blend_radius_m)
    movel([0.148063, -1.249196, -2.651763, -0.811430, 1.570796, 1.718859],accel_mss,speed_ms,0,blend_radius_m)
    movel([0.147607, -1.249561, -2.651569, -0.811259, 1.570796, 1.718403],accel_mss,speed_ms,0,blend_radius_m)
    movel([0.147376, -1.250034, -2.651316, -0.811039, 1.570796, 1.718172],accel_mss,speed_ms,0,blend_radius_m)
    movel([0.147470, -1.250406, -2.651117, -0.810865, 1.570796, 1.718267],accel_mss,speed_ms,0,blend_radius_m)
    movel([0.147850, -1.250512, -2.651061, -0.810816, 1.570796, 1.718646],accel_mss,speed_ms,0,blend_radius_m)
    movel([0.150091, -1.250076, -2.651294, -0.811019, 1.570796, 1.720887],accel_mss,speed_ms,0,blend_radius_m)
    movel([0.154750, -1.248766, -2.651992, -0.811631, 1.570796, 1.725547],accel_mss,speed_ms,0,blend_radius_m)
    movel([0.168985, -1.244516, -2.654243, -0.813630, 1.570796, 1.739782],accel_mss,speed_ms,0,blend_radius_m)
    movel([0.171897, -1.243658, -2.654695, -0.814036, 1.570796, 1.742693],accel_mss,speed_ms,0,blend_radius_m)
    speed_ms = 0.005
    movel([0.171897, -1.234190, -2.650078, -0.828122, 1.570796, 1.742693],accel_mss,speed_ms,0,blend_radius_m)
    speed_ms = 0.040
    movel([0.168490, -1.237774, -2.648209, -0.826406, 1.570796, 1.739287],accel_mss,speed_ms,0,blend_radius_m)
    speed_ms = 0.005
    movel([0.168490, -1.247226, -2.652810, -0.812353, 1.570796, 1.739287],accel_mss,speed_ms,0,blend_radius_m)
    speed_ms = 0.035
    movel([0.180881, -1.243620, -2.654715, -0.814054, 1.570796, 1.751678],accel_mss,speed_ms,0,blend_radius_m)
    movel([0.186532, -1.241910, -2.655613, -0.814866, 1.570796, 1.757329],accel_mss,speed_ms,0,blend_radius_m)
    movel([0.189878, -1.240794, -2.656197, -0.815398, 1.570796, 1.760674],accel_mss,speed_ms,0,blend_radius_m)
    movel([0.190250, -1.240542, -2.656329, -0.815518, 1.570796, 1.761047],accel_mss,speed_ms,0,blend_radius_m)
    movel([0.190455, -1.240171, -2.656522, -0.815696, 1.570796, 1.761251],accel_mss,speed_ms,0,blend_radius_m)
    movel([0.190386, -1.239876, -2.656676, -0.815837, 1.570796, 1.761182],accel_mss,speed_ms,0,blend_radius_m)
    movel([0.190077, -1.239814, -2.656709, -0.815866, 1.570796, 1.760873],accel_mss,speed_ms,0,blend_radius_m)
    movel([0.186805, -1.240549, -2.656325, -0.815515, 1.570796, 1.757601],accel_mss,speed_ms,0,blend_radius_m)
    movel([0.181191, -1.242029, -2.655551, -0.814810, 1.570796, 1.751988],accel_mss,speed_ms,0,blend_radius_m)
    movel([0.168787, -1.245601, -2.653670, -0.813117, 1.570796, 1.739583],accel_mss,speed_ms,0,blend_radius_m)
    movel([0.156400, -1.249324, -2.651695, -0.811370, 1.570796, 1.727197],accel_mss,speed_ms,0,blend_radius_m)
    movel([0.150774, -1.251149, -2.650720, -0.810519, 1.570796, 1.721570],accel_mss,speed_ms,0,blend_radius_m)
    movel([0.147454, -1.252349, -2.650078, -0.809963, 1.570796, 1.718251],accel_mss,speed_ms,0,blend_radius_m)
    movel([0.147092, -1.252605, -2.649940, -0.809844, 1.570796, 1.717888],accel_mss,speed_ms,0,blend_radius_m)
    movel([0.146904, -1.252970, -2.649744, -0.809675, 1.570796, 1.717700],accel_mss,speed_ms,0,blend_radius_m)
    movel([0.146988, -1.253250, -2.649594, -0.809545, 1.570796, 1.717784],accel_mss,speed_ms,0,blend_radius_m)
    movel([0.147302, -1.253297, -2.649568, -0.809524, 1.570796, 1.718098],accel_mss,speed_ms,0,blend_radius_m)
    movel([0.150556, -1.252474, -2.650011, -0.809905, 1.570796, 1.721352],accel_mss,speed_ms,0,blend_radius_m)
    movel([0.156135, -1.250885, -2.650862, -0.810642, 1.570796, 1.726931],accel_mss,speed_ms,0,blend_radius_m)
    movel([0.168490, -1.247226, -2.652810, -0.812353, 1.570796, 1.739287],accel_mss,speed_ms,0,blend_radius_m)
    movel([0.171393, -1.246372, -2.653263, -0.812754, 1.570796, 1.742190],accel_mss,speed_ms,0,blend_radius_m)
    speed_ms = 0.005
    movel([0.171393, -1.236916, -2.648658, -0.826815, 1.570796, 1.742190],accel_mss,speed_ms,0,blend_radius_m)
    speed_ms = 0.040
    movel([0.159403, -1.288678, -2.620008, -0.803703, 1.570796, 1.730199],accel_mss,speed_ms,0,blend_radius_m)
    speed_ms = 0.005
    movel([0.159403, -1.297872, -2.624380, -0.790137, 1.570796, 1.730199],accel_mss,speed_ms,0,blend_radius_m)
    speed_ms = 0.035
    movel([0.180242, -1.292350, -2.627635, -0.792403, 1.570796, 1.751038],accel_mss,speed_ms,0,blend_radius_m)
    movel([0.185199, -1.268162, -2.641443, -0.802785, 1.570796, 1.755995],accel_mss,speed_ms,0,blend_radius_m)
    movel([0.187829, -1.255340, -2.648468, -0.808581, 1.570796, 1.758625],accel_mss,speed_ms,0,blend_radius_m)
    movel([0.190058, -1.243366, -2.654849, -0.814174, 1.570796, 1.760855],accel_mss,speed_ms,0,blend_radius_m)
    movel([0.190007, -1.243068, -2.655005, -0.814316, 1.570796, 1.760803],accel_mss,speed_ms,0,blend_radius_m)
    movel([0.189757, -1.242935, -2.655075, -0.814379, 1.570796, 1.760554],accel_mss,speed_ms,0,blend_radius_m)
    movel([0.189184, -1.242993, -2.655044, -0.814351, 1.570796, 1.759980],accel_mss,speed_ms,0,blend_radius_m)
    movel([0.167590, -1.249144, -2.651791, -0.811454, 1.570796, 1.738386],accel_mss,speed_ms,0,blend_radius_m)
    movel([0.146189, -1.255715, -2.648265, -0.808409, 1.570796, 1.716985],accel_mss,speed_ms,0,blend_radius_m)
    movel([0.142308, -1.280153, -2.634690, -0.797546, 1.570796, 1.713104],accel_mss,speed_ms,0,blend_radius_m)
    movel([0.138633, -1.303685, -2.620910, -0.787795, 1.570796, 1.709430],accel_mss,speed_ms,0,blend_radius_m)
    movel([0.159403, -1.297872, -2.624380, -0.790137, 1.570796, 1.730199],accel_mss,speed_ms,0,blend_radius_m)
    movel([0.162141, -1.297128, -2.624820, -0.790440, 1.570796, 1.732937],accel_mss,speed_ms,0,blend_radius_m)
    speed_ms = 0.005
    movel([0.162141, -1.287930, -2.620446, -0.804013, 1.570796, 1.732937],accel_mss,speed_ms,0,blend_radius_m)
    speed_ms = 0.040
    movel([0.173092, -1.306432, -2.609414, -0.796543, 1.570796, 1.743888],accel_mss,speed_ms,0,blend_radius_m)
    speed_ms = 0.005
    movel([0.173092, -1.315524, -2.613706, -0.783159, 1.570796, 1.743888],accel_mss,speed_ms,0,blend_radius_m)
    speed_ms = 0.035
    movel([0.172750, -1.315473, -2.613738, -0.783179, 1.570796, 1.743547],accel_mss,speed_ms,0,blend_radius_m)
    movel([0.165825, -1.317133, -2.612712, -0.782543, 1.570796, 1.736621],accel_mss,speed_ms,0,blend_radius_m)
    movel([0.148824, -1.321500, -2.609999, -0.780889, 1.570796, 1.719620],accel_mss,speed_ms,0,blend_radius_m)
    movel([0.124966, -1.328113, -2.605842, -0.778433, 1.570796, 1.695762],accel_mss,speed_ms,0,blend_radius_m)
    movel([0.124236, -1.333290, -2.602547, -0.776552, 1.570796, 1.695032],accel_mss,speed_ms,0,blend_radius_m)
    movel([0.148189, -1.326585, -2.606808, -0.778996, 1.570796, 1.718985],accel_mss,speed_ms,0,blend_radius_m)
    movel([0.172245, -1.320262, -2.610771, -0.781356, 1.570796, 1.743042],accel_mss,speed_ms,0,blend_radius_m)
    movel([0.172824, -1.318024, -2.612161, -0.782204, 1.570796, 1.743620],accel_mss,speed_ms,0,blend_radius_m)
    movel([0.173142, -1.316362, -2.613189, -0.782838, 1.570796, 1.743939],accel_mss,speed_ms,0,blend_radius_m)
    movel([0.173183, -1.315740, -2.613573, -0.783076, 1.570796, 1.743979],accel_mss,speed_ms,0,blend_radius_m)
    movel([0.173092, -1.315524, -2.613706, -0.783159, 1.570796, 1.743888],accel_mss,speed_ms,0,blend_radius_m)
    movel([0.172750, -1.315473, -2.613738, -0.783179, 1.570796, 1.743547],accel_mss,speed_ms,0,blend_radius_m)
    movel([0.170483, -1.316012, -2.613405, -0.782972, 1.570796, 1.741279],accel_mss,speed_ms,0,blend_radius_m)
    speed_ms = 0.005
    movel([0.170483, -1.306923, -2.609116, -0.796351, 1.570796, 1.741279],accel_mss,speed_ms,0,blend_radius_m)
    speed_ms = 0.040
    movel([0.171885, -1.312776, -2.605530, -0.794083, 1.570796, 1.742681],accel_mss,speed_ms,0,blend_radius_m)
    speed_ms = 0.005
    movel([0.171885, -1.321830, -2.609794, -0.780766, 1.570796, 1.742681],accel_mss,speed_ms,0,blend_radius_m)
    speed_ms = 0.035
    movel([0.171545, -1.321781, -2.609824, -0.780784, 1.570796, 1.742342],accel_mss,speed_ms,0,blend_radius_m)
    movel([0.164662, -1.323416, -2.608801, -0.780172, 1.570796, 1.735458],accel_mss,speed_ms,0,blend_radius_m)
    movel([0.147766, -1.327716, -2.606094, -0.778579, 1.570796, 1.718562],accel_mss,speed_ms,0,blend_radius_m)
    movel([0.124053, -1.334231, -2.601945, -0.776214, 1.570796, 1.694849],accel_mss,speed_ms,0,blend_radius_m)
    movel([0.123616, -1.339493, -2.598551, -0.774345, 1.570796, 1.694412],accel_mss,speed_ms,0,blend_radius_m)
    movel([0.147241, -1.333059, -2.602695, -0.776635, 1.570796, 1.718037],accel_mss,speed_ms,0,blend_radius_m)
    movel([0.170960, -1.327003, -2.606545, -0.778842, 1.570796, 1.741756],accel_mss,speed_ms,0,blend_radius_m)
    movel([0.171576, -1.324546, -2.608092, -0.779751, 1.570796, 1.742373],accel_mss,speed_ms,0,blend_radius_m)
    movel([0.171923, -1.322733, -2.609229, -0.780427, 1.570796, 1.742719],accel_mss,speed_ms,0,blend_radius_m)
    movel([0.171974, -1.322054, -2.609654, -0.780682, 1.570796, 1.742770],accel_mss,speed_ms,0,blend_radius_m)
    movel([0.171885, -1.321830, -2.609794, -0.780766, 1.570796, 1.742681],accel_mss,speed_ms,0,blend_radius_m)
    movel([0.171545, -1.321781, -2.609824, -0.780784, 1.570796, 1.742342],accel_mss,speed_ms,0,blend_radius_m)
    movel([0.169295, -1.322311, -2.609493, -0.780585, 1.570796, 1.740091],accel_mss,speed_ms,0,blend_radius_m)
    speed_ms = 0.005
    movel([0.169295, -1.313260, -2.605232, -0.793897, 1.570796, 1.740091],accel_mss,speed_ms,0,blend_radius_m)
    speed_ms = 0.040
    movel([0.170695, -1.319062, -2.601629, -0.791697, 1.570796, 1.741491],accel_mss,speed_ms,0,blend_radius_m)
    speed_ms = 0.005
    movel([0.170695, -1.328078, -2.605865, -0.778446, 1.570796, 1.741491],accel_mss,speed_ms,0,blend_radius_m)
    speed_ms = 0.035
    movel([0.170358, -1.328027, -2.605897, -0.778465, 1.570796, 1.741154],accel_mss,speed_ms,0,blend_radius_m)
    movel([0.163531, -1.329632, -2.604879, -0.777877, 1.570796, 1.734328],accel_mss,speed_ms,0,blend_radius_m)
    movel([0.146775, -1.333858, -2.602184, -0.776348, 1.570796, 1.717571],accel_mss,speed_ms,0,blend_radius_m)
    movel([0.123257, -1.340261, -2.598052, -0.774075, 1.570796, 1.694053],accel_mss,speed_ms,0,blend_radius_m)
    movel([0.122546, -1.345342, -2.594735, -0.772312, 1.570796, 1.693343],accel_mss,speed_ms,0,blend_radius_m)
    movel([0.146160, -1.338846, -2.598970, -0.774573, 1.570796, 1.716956],accel_mss,speed_ms,0,blend_radius_m)
    movel([0.169873, -1.332724, -2.602909, -0.776756, 1.570796, 1.740669],accel_mss,speed_ms,0,blend_radius_m)
    movel([0.170437, -1.330530, -2.604309, -0.777551, 1.570796, 1.741233],accel_mss,speed_ms,0,blend_radius_m)
    movel([0.170747, -1.328901, -2.605343, -0.778145, 1.570796, 1.741543],accel_mss,speed_ms,0,blend_radius_m)
    movel([0.170785, -1.328291, -2.605730, -0.778368, 1.570796, 1.741581],accel_mss,speed_ms,0,blend_radius_m)
    movel([0.170695, -1.328078, -2.605865, -0.778446, 1.570796, 1.741491],accel_mss,speed_ms,0,blend_radius_m)
    movel([0.170358, -1.328027, -2.605897, -0.778465, 1.570796, 1.741154],accel_mss,speed_ms,0,blend_radius_m)
    movel([0.168123, -1.328548, -2.605567, -0.778274, 1.570796, 1.738919],accel_mss,speed_ms,0,blend_radius_m)
    speed_ms = 0.005
    movel([0.168123, -1.319535, -2.601334, -0.791520, 1.570796, 1.738919],accel_mss,speed_ms,0,blend_radius_m)
    speed_ms = 0.040
    movel([0.189326, -1.316554, -2.603192, -0.792643, 1.570796, 1.760122],accel_mss,speed_ms,0,blend_radius_m)
    speed_ms = 0.005
    movel([0.189326, -1.325585, -2.607438, -0.779365, 1.570796, 1.760122],accel_mss,speed_ms,0,blend_radius_m)
    speed_ms = 0.035
    movel([0.180592, -1.327517, -2.606220, -0.778652, 1.570796, 1.751388],accel_mss,speed_ms,0,blend_radius_m)
    movel([0.177754, -1.328068, -2.605871, -0.778450, 1.570796, 1.748550],accel_mss,speed_ms,0,blend_radius_m)
    movel([0.177568, -1.327903, -2.605976, -0.778511, 1.570796, 1.748364],accel_mss,speed_ms,0,blend_radius_m)
    movel([0.177841, -1.327627, -2.606150, -0.778612, 1.570796, 1.748637],accel_mss,speed_ms,0,blend_radius_m)
    movel([0.184450, -1.325835, -2.607281, -0.779273, 1.570796, 1.755246],accel_mss,speed_ms,0,blend_radius_m)
    movel([0.189528, -1.324620, -2.608046, -0.779723, 1.570796, 1.760325],accel_mss,speed_ms,0,blend_radius_m)
    movel([0.198276, -1.322741, -2.609224, -0.780424, 1.570796, 1.769072],accel_mss,speed_ms,0,blend_radius_m)
    movel([0.201118, -1.322233, -2.609541, -0.780614, 1.570796, 1.771914],accel_mss,speed_ms,0,blend_radius_m)
    movel([0.201298, -1.322406, -2.609434, -0.780550, 1.570796, 1.772094],accel_mss,speed_ms,0,blend_radius_m)
    movel([0.201019, -1.322680, -2.609262, -0.780447, 1.570796, 1.771815],accel_mss,speed_ms,0,blend_radius_m)
    movel([0.194401, -1.324393, -2.608188, -0.779808, 1.570796, 1.765197],accel_mss,speed_ms,0,blend_radius_m)
    movel([0.189326, -1.325585, -2.607438, -0.779365, 1.570796, 1.760122],accel_mss,speed_ms,0,blend_radius_m)
    movel([0.186699, -1.326160, -2.607077, -0.779153, 1.570796, 1.757495],accel_mss,speed_ms,0,blend_radius_m)
    speed_ms = 0.005
    movel([0.186699, -1.317132, -2.602833, -0.792424, 1.570796, 1.757495],accel_mss,speed_ms,0,blend_radius_m)
    speed_ms = 0.040
    movel([0.189731, -1.314611, -2.604397, -0.793381, 1.570796, 1.760527],accel_mss,speed_ms,0,blend_radius_m)
    speed_ms = 0.005
    movel([0.189731, -1.323653, -2.608652, -0.780083, 1.570796, 1.760527],accel_mss,speed_ms,0,blend_radius_m)
    speed_ms = 0.035
    movel([0.183077, -1.325192, -2.607686, -0.779511, 1.570796, 1.753873],accel_mss,speed_ms,0,blend_radius_m)
    movel([0.179988, -1.325829, -2.607285, -0.779275, 1.570796, 1.750785],accel_mss,speed_ms,0,blend_radius_m)
    movel([0.178290, -1.326057, -2.607142, -0.779191, 1.570796, 1.749086],accel_mss,speed_ms,0,blend_radius_m)
    movel([0.178048, -1.325982, -2.607188, -0.779218, 1.570796, 1.748844],accel_mss,speed_ms,0,blend_radius_m)
    movel([0.177995, -1.325743, -2.607339, -0.779307, 1.570796, 1.748791],accel_mss,speed_ms,0,blend_radius_m)
    movel([0.178152, -1.325453, -2.607522, -0.779414, 1.570796, 1.748949],accel_mss,speed_ms,0,blend_radius_m)
    movel([0.178450, -1.325249, -2.607650, -0.779490, 1.570796, 1.749246],accel_mss,speed_ms,0,blend_radius_m)
    movel([0.180226, -1.324640, -2.608033, -0.779716, 1.570796, 1.751022],accel_mss,speed_ms,0,blend_radius_m)
    movel([0.183361, -1.323793, -2.608565, -0.780031, 1.570796, 1.754157],accel_mss,speed_ms,0,blend_radius_m)
    movel([0.190036, -1.322200, -2.609562, -0.780627, 1.570796, 1.760832],accel_mss,speed_ms,0,blend_radius_m)
    movel([0.196704, -1.320689, -2.610506, -0.781195, 1.570796, 1.767501],accel_mss,speed_ms,0,blend_radius_m)
    movel([0.199800, -1.320087, -2.610880, -0.781422, 1.570796, 1.770596],accel_mss,speed_ms,0,blend_radius_m)
    movel([0.201499, -1.319889, -2.611004, -0.781497, 1.570796, 1.772295],accel_mss,speed_ms,0,blend_radius_m)
    movel([0.201737, -1.319970, -2.610953, -0.781466, 1.570796, 1.772534],accel_mss,speed_ms,0,blend_radius_m)
    movel([0.201784, -1.320215, -2.610801, -0.781374, 1.570796, 1.772580],accel_mss,speed_ms,0,blend_radius_m)
    movel([0.201618, -1.320506, -2.610619, -0.781263, 1.570796, 1.772415],accel_mss,speed_ms,0,blend_radius_m)
    movel([0.201317, -1.320708, -2.610493, -0.781187, 1.570796, 1.772114],accel_mss,speed_ms,0,blend_radius_m)
    movel([0.199535, -1.321291, -2.610130, -0.780968, 1.570796, 1.770331],accel_mss,speed_ms,0,blend_radius_m)
    movel([0.196399, -1.322099, -2.609626, -0.780665, 1.570796, 1.767195],accel_mss,speed_ms,0,blend_radius_m)
    movel([0.189731, -1.323653, -2.608652, -0.780083, 1.570796, 1.760527],accel_mss,speed_ms,0,blend_radius_m)
    movel([0.187092, -1.324259, -2.608272, -0.779857, 1.570796, 1.757888],accel_mss,speed_ms,0,blend_radius_m)
    speed_ms = 0.005
    movel([0.187092, -1.315220, -2.604020, -0.793149, 1.570796, 1.757888],accel_mss,speed_ms,0,blend_radius_m)
    speed_ms = 0.040
    movel([0.190239, -1.312172, -2.605902, -0.794315, 1.570796, 1.761036],accel_mss,speed_ms,0,blend_radius_m)
    speed_ms = 0.005
    movel([0.190239, -1.321230, -2.610168, -0.780991, 1.570796, 1.761036],accel_mss,speed_ms,0,blend_radius_m)
    speed_ms = 0.035
    movel([0.196926, -1.319665, -2.611142, -0.781581, 1.570796, 1.767722],accel_mss,speed_ms,0,blend_radius_m)
    movel([0.200071, -1.318852, -2.611648, -0.781889, 1.570796, 1.770868],accel_mss,speed_ms,0,blend_radius_m)
    movel([0.201858, -1.318266, -2.612011, -0.782112, 1.570796, 1.772655],accel_mss,speed_ms,0,blend_radius_m)
    movel([0.202160, -1.318064, -2.612136, -0.782189, 1.570796, 1.772957],accel_mss,speed_ms,0,blend_radius_m)
    movel([0.202326, -1.317771, -2.612318, -0.782300, 1.570796, 1.773123],accel_mss,speed_ms,0,blend_radius_m)
    movel([0.202280, -1.317525, -2.612470, -0.782394, 1.570796, 1.773076],accel_mss,speed_ms,0,blend_radius_m)
    movel([0.202041, -1.317444, -2.612520, -0.782425, 1.570796, 1.772837],accel_mss,speed_ms,0,blend_radius_m)
    movel([0.200337, -1.317644, -2.612396, -0.782348, 1.570796, 1.771133],accel_mss,speed_ms,0,blend_radius_m)
    movel([0.197233, -1.318250, -2.612021, -0.782118, 1.570796, 1.768030],accel_mss,speed_ms,0,blend_radius_m)
    movel([0.190546, -1.319771, -2.611077, -0.781541, 1.570796, 1.761342],accel_mss,speed_ms,0,blend_radius_m)
    movel([0.183852, -1.321374, -2.610078, -0.780937, 1.570796, 1.754649],accel_mss,speed_ms,0,blend_radius_m)
    movel([0.180709, -1.322227, -2.609546, -0.780617, 1.570796, 1.751505],accel_mss,speed_ms,0,blend_radius_m)
    movel([0.178927, -1.322838, -2.609163, -0.780388, 1.570796, 1.749724],accel_mss,speed_ms,0,blend_radius_m)
    movel([0.178629, -1.323044, -2.609034, -0.780311, 1.570796, 1.749426],accel_mss,speed_ms,0,blend_radius_m)
    movel([0.178471, -1.323335, -2.608852, -0.780202, 1.570796, 1.749267],accel_mss,speed_ms,0,blend_radius_m)
    movel([0.178524, -1.323575, -2.608702, -0.780113, 1.570796, 1.749321],accel_mss,speed_ms,0,blend_radius_m)
    movel([0.178766, -1.323649, -2.608655, -0.780085, 1.570796, 1.749563],accel_mss,speed_ms,0,blend_radius_m)
    movel([0.180470, -1.323420, -2.608799, -0.780170, 1.570796, 1.751266],accel_mss,speed_ms,0,blend_radius_m)
    movel([0.183567, -1.322778, -2.609201, -0.780410, 1.570796, 1.754363],accel_mss,speed_ms,0,blend_radius_m)
    movel([0.190239, -1.321230, -2.610168, -0.780991, 1.570796, 1.761036],accel_mss,speed_ms,0,blend_radius_m)
    movel([0.192890, -1.320606, -2.610557, -0.781226, 1.570796, 1.763687],accel_mss,speed_ms,0,blend_radius_m)
    speed_ms = 0.005
    movel([0.192890, -1.311544, -2.606288, -0.794556, 1.570796, 1.763687],accel_mss,speed_ms,0,blend_radius_m)
    speed_ms = 0.040
    movel([0.190322, -1.309359, -2.607629, -0.795401, 1.570796, 1.761118],accel_mss,speed_ms,0,blend_radius_m)
    speed_ms = 0.005
    movel([0.190322, -1.318434, -2.611907, -0.782048, 1.570796, 1.761118],accel_mss,speed_ms,0,blend_radius_m)
    speed_ms = 0.035
    movel([0.202817, -1.315563, -2.613682, -0.783144, 1.570796, 1.773614],accel_mss,speed_ms,0,blend_radius_m)
    movel([0.204528, -1.307899, -2.618366, -0.786123, 1.570796, 1.775324],accel_mss,speed_ms,0,blend_radius_m)
    movel([0.206268, -1.300139, -2.623031, -0.789218, 1.570796, 1.777065],accel_mss,speed_ms,0,blend_radius_m)
    movel([0.193884, -1.303048, -2.621292, -0.788049, 1.570796, 1.764681],accel_mss,speed_ms,0,blend_radius_m)
    movel([0.181516, -1.306068, -2.619474, -0.786847, 1.570796, 1.752313],accel_mss,speed_ms,0,blend_radius_m)
    movel([0.180967, -1.307264, -2.618751, -0.786374, 1.570796, 1.751764],accel_mss,speed_ms,0,blend_radius_m)
    movel([0.180691, -1.308031, -2.618286, -0.786072, 1.570796, 1.751488],accel_mss,speed_ms,0,blend_radius_m)
    movel([0.179122, -1.314971, -2.614047, -0.783372, 1.570796, 1.749918],accel_mss,speed_ms,0,blend_radius_m)
    movel([0.177840, -1.321418, -2.610051, -0.780920, 1.570796, 1.748636],accel_mss,speed_ms,0,blend_radius_m)
    movel([0.190322, -1.318434, -2.611907, -0.782048, 1.570796, 1.761118],accel_mss,speed_ms,0,blend_radius_m)
    movel([0.192980, -1.317813, -2.612292, -0.782284, 1.570796, 1.763776],accel_mss,speed_ms,0,blend_radius_m)
    speed_ms = 0.005
    movel([0.192980, -1.308735, -2.608010, -0.795644, 1.570796, 1.763776],accel_mss,speed_ms,0,blend_radius_m)
    speed_ms = 0.040
    movel([0.193546, -1.291298, -2.618470, -0.802621, 1.570796, 1.764342],accel_mss,speed_ms,0,blend_radius_m)
    speed_ms = 0.005
    movel([0.193546, -1.300477, -2.622830, -0.789082, 1.570796, 1.764342],accel_mss,speed_ms,0,blend_radius_m)
    speed_ms = 0.035
    movel([0.193910, -1.299720, -2.623281, -0.789388, 1.570796, 1.764706],accel_mss,speed_ms,0,blend_radius_m)
    movel([0.194146, -1.298971, -2.623727, -0.789691, 1.570796, 1.764942],accel_mss,speed_ms,0,blend_radius_m)
    movel([0.196571, -1.287547, -2.630436, -0.794406, 1.570796, 1.767367],accel_mss,speed_ms,0,blend_radius_m)
    movel([0.196568, -1.287181, -2.630648, -0.794560, 1.570796, 1.767365],accel_mss,speed_ms,0,blend_radius_m)
    movel([0.196402, -1.286911, -2.630804, -0.794673, 1.570796, 1.767198],accel_mss,speed_ms,0,blend_radius_m)
    movel([0.196111, -1.286854, -2.630837, -0.794697, 1.570796, 1.766907],accel_mss,speed_ms,0,blend_radius_m)
    movel([0.190413, -1.288077, -2.630128, -0.794184, 1.570796, 1.761209],accel_mss,speed_ms,0,blend_radius_m)
    movel([0.184721, -1.289516, -2.629291, -0.793581, 1.570796, 1.755517],accel_mss,speed_ms,0,blend_radius_m)
    movel([0.183242, -1.296857, -2.624981, -0.790551, 1.570796, 1.754038],accel_mss,speed_ms,0,blend_radius_m)
    movel([0.181787, -1.304113, -2.620652, -0.787624, 1.570796, 1.752583],accel_mss,speed_ms,0,blend_radius_m)
    movel([0.187417, -1.302720, -2.621489, -0.788181, 1.570796, 1.758213],accel_mss,speed_ms,0,blend_radius_m)
    movel([0.190438, -1.301953, -2.621948, -0.788488, 1.570796, 1.761235],accel_mss,speed_ms,0,blend_radius_m)
    movel([0.192066, -1.301442, -2.622254, -0.788693, 1.570796, 1.762862],accel_mss,speed_ms,0,blend_radius_m)
    movel([0.193028, -1.300988, -2.622525, -0.788876, 1.570796, 1.763825],accel_mss,speed_ms,0,blend_radius_m)
    movel([0.193546, -1.300477, -2.622830, -0.789082, 1.570796, 1.764342],accel_mss,speed_ms,0,blend_radius_m)
    movel([0.193910, -1.299720, -2.623281, -0.789388, 1.570796, 1.764706],accel_mss,speed_ms,0,blend_radius_m)
    movel([0.194146, -1.298971, -2.623727, -0.789691, 1.570796, 1.764942],accel_mss,speed_ms,0,blend_radius_m)
    movel([0.194366, -1.297922, -2.624350, -0.790117, 1.570796, 1.765163],accel_mss,speed_ms,0,blend_radius_m)
    speed_ms = 0.005
    movel([0.194366, -1.288728, -2.619979, -0.803682, 1.570796, 1.765163],accel_mss,speed_ms,0,blend_radius_m)
    speed_ms = 0.040
    movel([0.200796, -1.290318, -2.619046, -0.803024, 1.570796, 1.771592],accel_mss,speed_ms,0,blend_radius_m)
    speed_ms = 0.005
    movel([0.200796, -1.299503, -2.623410, -0.789476, 1.570796, 1.771592],accel_mss,speed_ms,0,blend_radius_m)
    speed_ms = 0.035
    movel([0.194871, -1.300911, -2.622571, -0.788907, 1.570796, 1.765668],accel_mss,speed_ms,0,blend_radius_m)
    movel([0.196504, -1.293697, -2.626845, -0.791847, 1.570796, 1.767300],accel_mss,speed_ms,0,blend_radius_m)
    movel([0.198164, -1.286398, -2.631101, -0.794889, 1.570796, 1.768960],accel_mss,speed_ms,0,blend_radius_m)
    movel([0.203393, -1.284986, -2.631917, -0.795486, 1.570796, 1.774189],accel_mss,speed_ms,0,blend_radius_m)
    movel([0.208814, -1.283705, -2.632655, -0.796029, 1.570796, 1.779610],accel_mss,speed_ms,0,blend_radius_m)
    movel([0.209297, -1.283684, -2.632667, -0.796038, 1.570796, 1.780093],accel_mss,speed_ms,0,blend_radius_m)
    movel([0.209502, -1.283789, -2.632606, -0.795993, 1.570796, 1.780299],accel_mss,speed_ms,0,blend_radius_m)
    movel([0.209575, -1.284009, -2.632480, -0.795900, 1.570796, 1.780371],accel_mss,speed_ms,0,blend_radius_m)
    movel([0.209473, -1.285300, -2.631736, -0.795353, 1.570796, 1.780269],accel_mss,speed_ms,0,blend_radius_m)
    movel([0.209113, -1.287403, -2.630519, -0.794467, 1.570796, 1.779909],accel_mss,speed_ms,0,blend_radius_m)
    movel([0.206722, -1.298121, -2.624232, -0.790036, 1.570796, 1.777519],accel_mss,speed_ms,0,blend_radius_m)
    movel([0.200796, -1.299503, -2.623410, -0.789476, 1.570796, 1.771592],accel_mss,speed_ms,0,blend_radius_m)
    movel([0.198084, -1.300144, -2.623028, -0.789216, 1.570796, 1.768880],accel_mss,speed_ms,0,blend_radius_m)
    speed_ms = 0.005
    movel([0.198084, -1.256176, -2.600655, -0.855558, 1.570796, 1.768880],accel_mss,speed_ms,0,blend_radius_m)
    speed_ms = 1.000
    movel([0.198084, -1.166121, -2.539164, -1.007104, 1.570796, 1.768880],accel_mss,speed_ms,0,blend_radius_m)
    # End of main program
  end

  Machining3()
end
